// TwinCAT 3 PLC project ProtoSimPLC
// ProgramVersion: 3.1.4022.3
// libraries:
//   Tc2_Standard, * (Beckhoff Automation GmbH)
//   Tc2_System, * (Beckhoff Automation GmbH)
//   Tc3_Module, * (Beckhoff Automation GmbH)
//   Vacuum System Simulator Library, * (SLAC)
// project tree:
//   GVLs/ GVL_VARIABLES.TcGVL, GVL_DEVICES.TcGVL
//   POUs/ MAIN.TcPOU, PRG_HEARTBEAT.TcPOU, PRG_OverridePressure.TcPOU, PRG_SIMULATION.TcPOU
//   / SimTask.TcTTO
// (motion and I/O tree: see PLC project xtessxrplc)
// real-time tasks:
//   TASK PlcTask: cycle T#10ms, priority 20, ADS port 350
//   TASK SimTask: cycle T#5ms, priority 21, ADS port 351
// variable links:
//   ProtoSimPLC/ProtoSimPLC Instance <-> Device 2 (EtherCAT Simulation)/=+-A1
//     SimTask Outputs/GVL_DEVICES.stVgc_MR1K4_VGC_1.q_xClsLS <-> Channel 4/Input
//     SimTask Outputs/GVL_DEVICES.stVgc_MR1K4_VGC_1.q_xOpnLS <-> Channel 3/Input
//     SimTask Outputs/GVL_DEVICES.stVgc_TV2K4_VGC_1.q_xClsLS <-> Channel 8/Input
//     SimTask Outputs/GVL_DEVICES.stVgc_TV2K4_VGC_1.q_xOpnLS <-> Channel 7/Input
//     SimTask Inputs/GVL_DEVICES.stVgc_MR1K4_VGC_1.i_xSol <-> Channel 9/Output
//     SimTask Inputs/GVL_DEVICES.stVgc_TV2K4_VGC_1.i_xSol <-> Channel 13/Output
//   ProtoSimPLC/ProtoSimPLC Instance <-> Device 2 (EtherCAT Simulation)/=+-A2
//     SimTask Outputs/GVL_DEVICES.stMks500_TV2K4_GCC_1.q_iRawPress <-> AI Standard Channel 1/Value
//     SimTask Outputs/GVL_DEVICES.stMks275_TV2K4_GPI_1.q_iRawPress <-> AI Standard Channel 4/Value
//   ProtoSimPLC/ProtoSimPLC Instance <-> Device 2 (EtherCAT Simulation)/=+-A3
//     SimTask Inputs/GVL_DEVICES.stMks500_TV2K4_GCC_1.i_xHvOn <-> Channel 1/Output
//   ProtoSimPLC/ProtoSimPLC Instance <-> Device 2 (EtherCAT Simulation)/=+-DO1
//     SimTask Inputs/GVL_DEVICES.stGamPip_TV2KO_PIP_1.xOn <-> Channel 1/Output

CONFIGURATION ProtoSimPLC
    RESOURCE PLC ON TwinCAT3
        TASK SimTask(INTERVAL := T#5ms, PRIORITY := 21);
        PROGRAM PRG_HEARTBEAT WITH SimTask : PRG_HEARTBEAT;
        PROGRAM MAIN WITH SimTask : MAIN;
    END_RESOURCE
END_CONFIGURATION

// ---- GVLs/GVL_VARIABLES.TcGVL
VAR_GLOBAL
END_VAR

// ---- GVLs/GVL_DEVICES.TcGVL
VAR_GLOBAL
	
	Global_Leak	: REAL := 0;
	Global_Pressure : REAL := 0.0079;
	New_Pressure : REAL := 22.0; //Torr
	Global_OverridePressure	: BOOL := FALSE;//initially set to be false

	// volumes
	
	stVl_Start : ST_Volume := (
		rVolume := 1E3, 
		rPressure := Global_Pressure, 
		rVLeak := Global_Leak
		);
	
	stVl_Proto : ST_Volume := (
		rVolume := 1E3, 
		rPressure := Global_Pressure, 
		rVLeak := Global_Leak
		);
		
	stVl_End : ST_Volume := (
		rVolume := 1E3, 
		rPressure := Global_Pressure, 
		rVLeak := Global_Leak
		);
	
	// valves
	
	stVgc_TV2K4_VGC_1 : ST_VacuumValve := (q_xClsLS := TRUE, q_xOpnLS := FALSE); // VV9S
	stVgc_MR1K4_VGC_1 : ST_VacuumValve := (q_xClsLS := TRUE, q_xOpnLS := FALSE); // VV10S
	
	fbVgc_TV2K4_VGC_1 : FB_VacuumValve; // VV9S
	fbVgc_MR1K4_VGC_1 : FB_VacuumValve; // VV10S
	
	// gauges	
	
	stMks275_MR2K3_GPI_1 : ST_MKS_275 := (q_xGaugeConnected := TRUE);
	stMks275_TV2K4_GPI_1 : ST_MKS_275 := (q_xGaugeConnected := TRUE);
	stMks275_MR1K4_GPI_1 : ST_MKS_275 := (q_xGaugeConnected := TRUE);
	stMks500_MR2K3_GCC_1 : ST_MKS_500 := (q_xGaugeConnected := TRUE);
	stMks500_TV2K4_GCC_1 : ST_MKS_500 := (q_xGaugeConnected := TRUE);
	stMks500_MR1K4_GCC_1 : ST_MKS_500 := (q_xGaugeConnected := TRUE);

	fbMks275_MR2K3_GPI_1 : FB_MKS_275;
	fbMks275_TV2K4_GPI_1 : FB_MKS_275;
	fbMks275_MR1K4_GPI_1 : FB_MKS_275;
	fbMks500_MR2K3_GCC_1 : FB_MKS_500;
	fbMks500_TV2K4_GCC_1 : FB_MKS_500;
	fbMks500_MR1K4_GCC_1 : FB_MKS_500;

	// pumps
	
	stGamPip_TV2KO_PIP_1 : ST_GAM_PIP;
	
	fbGamPip_TV2KO_PIP_1 : FB_GAM_PIP;

END_VAR

// ---- POUs/PRG_HEARTBEAT.TcPOU
PROGRAM PRG_HEARTBEAT
VAR
	heartbeat AT %Q* : UINT := 0;
END_VAR

heartbeat := heartbeat + 1;
IF heartbeat > 65000
	THEN heartbeat := 0;
END_IF

END_PROGRAM

// ---- POUs/MAIN.TcPOU
PROGRAM MAIN
VAR
END_VAR

PRG_HEARTBEAT();
PRG_OverridePressure();
PRG_SIMULATION();

END_PROGRAM

// ---- POUs/PRG_OverridePressure.TcPOU
PROGRAM PRG_OverridePressure
VAR
	fb_SetPressure : FB_SetChamberPressure; 
END_VAR

fb_SetPressure(chamber := stVl_Proto, rNewPressure := New_Pressure, Override:= Global_OverridePressure);

END_PROGRAM

// ---- POUs/PRG_SIMULATION.TcPOU
PROGRAM PRG_SIMULATION
VAR
END_VAR

// valves

fbVgc_TV2K4_VGC_1(
	stAVol := stVl_Start,
	stBvol := stVl_Proto,
	stValve := stVgc_TV2K4_VGC_1
	); // VV9S
	
fbVgc_MR1K4_VGC_1(
	stAVol := stVl_Proto,
	stBvol := stVl_End,
	stValve := stVgc_MR1K4_VGC_1
	); // VV10S

// gauges

fbMks275_TV2K4_GPI_1(stVolume := stVl_Proto, stGauge:= stMks275_TV2K4_GPI_1);
fbMks500_TV2K4_GCC_1(stVolume := stVl_Proto, stGauge:= stMks500_TV2K4_GCC_1);

// pumps

fbGamPip_TV2KO_PIP_1(stVolume := stVl_Proto, stPip := stGamPip_TV2KO_PIP_1);

END_PROGRAM
